PROGRAM PG_AlarmHistory
VAR
	i:UDINT;
	AlarmHistoryData_Write:ST_AlarmInfo_DB_save;
	
	bWriteResult: ARRAY[0..GVL.Max_IndexNum-1] OF BOOL;
	
	repeatTimer:TON;
	writeFailCount:UDINT;
END_VAR


//simulate that Peak Data amount as 500 ms
repeatTimer(IN:=TRUE,PT:=T#300MS);

IF repeatTimer.Q THEN
	
	repeatTimer(in:=FALSE);
	
	//simulate Peak save data amount
	FOR i:=0 TO GVL.Max_IndexNum-1 DO
		bWriteResult[i]:=GVL.fbDataToNovRam[i].M_AlarmHistory(addData:=AlarmHistoryData_Write);
		
		IF bWriteResult[i]=FALSE THEN
			writeFailCount:=writeFailCount+1;
		END_IF
	END_FOR
	
END_IF

END_PROGRAM

(* stored: Version 1.1.0.1, ProductVersion 3.1.4024.11
   POU PG_AlarmHistory: Id {54f410b2-b83a-4d7a-938e-1ab226b5f3f6}, SpecialFunc None *)
